// TIA Portal V17 export
// export: Created 2022-12-02T11:58:37.0501508Z, ExportSetting WithDefaults, DisplayName Totally Integrated Automation Portal, DisplayVersion V17 Update 3, DisplayName TIA Portal Openness, DisplayVersion V17 Update 3, DisplayName TIA Portal Version Control Interface, DisplayVersion V17, DisplayName STEP 7 Professional, DisplayVersion V17 Update 3, DisplayName STEP 7 Safety, DisplayVersion V17, DisplayName WinCC Advanced, DisplayVersion V17 Update 3
FUNCTION "Block_1" : Void   // FC2, LAD
{ S7_Optimized_Access := 'TRUE' }
VERSION : 0.1
// stored: AutoNumber true, IsIECCheckEnabled false, SetENOAutomatically false, UDAEnableTagReadback false
   VAR_INPUT
      mmm : Bool;
   END_VAR
   VAR_OUTPUT
      siuu : Bool;
   END_VAR
BEGIN

REGION Network 1
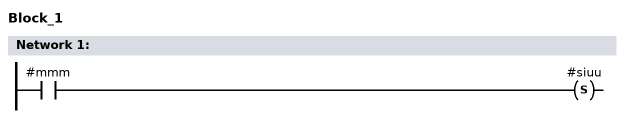
   RUNG wire#powerrail
      Contact( #mmm )
      S_Coil( #siuu )
   END_RUNG
   // the same network as SCL:
   IF #mmm THEN #siuu := TRUE; END_IF;
END_REGION
END_FUNCTION
